// TwinCAT 3 PLC project Nepionic_PackML
// Title: Nepionic_PackML
// Company: Nepionic
// Author: Nepionic
// ProjectVersion: 0.1.0
// ProgramVersion: 3.1.4026.19
// libraries:
//   Tc2_System, * (Beckhoff Automation GmbH)
// project tree:
//   Commands/ AbortedCommands.TcIO, AbortingCommands.TcIO, ClearingCommands.TcIO, CompletedCommands.TcIO, CompletingCommands.TcIO, ExecuteCommands.TcIO, HeldCommands.TcIO, HoldingCommands.TcIO, IdleCommands.TcIO, ResettingCommands.TcIO, StartingCommands.TcIO, StoppedCommands.TcIO, StoppingCommands.TcIO, SuspendedCommands.TcIO, SuspendingCommands.TcIO, UnholdingCommands.TcIO, UnsuspendingCommands.TcIO
//   StateMachine/ State.TcDUT, StateMachine.TcPOU
//   UnitMode/ UnitMode.TcIO (not stored), DefaultUnitMode.TcPOU

// ---- StateMachine/State.TcDUT
{attribute 'qualified_only'}
{attribute 'strict'}
TYPE State :
(
	UNDEFINED := 0,
    CLEARING := 1,
    STOPPED := 2,
    STARTING := 3,
    IDLE := 4,
    SUSPENDED := 5,
	EXECUTE := 6,
    STOPPING := 7,
    ABORTING := 8,
    ABORTED := 9,
    HOLDING := 10,
    HELD := 11,
    UNHOLDING := 12,
    SUSPENDING := 13,
    UNSUSPENDING := 14,
    RESETTING := 15,
    COMPLETING := 16,
    COMPLETE := 17
);
END_TYPE

// ---- Commands/AbortedCommands.TcIO
INTERFACE PUBLIC AbortedCommands

METHOD PUBLIC Clear
END_METHOD

END_INTERFACE

// ---- Commands/AbortingCommands.TcIO
INTERFACE PUBLIC AbortingCommands

METHOD PUBLIC StateComplete
END_METHOD

END_INTERFACE

// ---- Commands/ClearingCommands.TcIO
INTERFACE PUBLIC ClearingCommands

METHOD PUBLIC Abort
END_METHOD

METHOD PUBLIC StateComplete
END_METHOD

END_INTERFACE

// ---- Commands/CompletedCommands.TcIO
INTERFACE PUBLIC CompletedCommands

METHOD PUBLIC Abort
END_METHOD

METHOD PUBLIC Reset
END_METHOD

METHOD PUBLIC Stop
END_METHOD

END_INTERFACE

// ---- Commands/CompletingCommands.TcIO
INTERFACE PUBLIC CompletingCommands

METHOD PUBLIC Abort
END_METHOD

METHOD PUBLIC StateComplete
END_METHOD

METHOD PUBLIC Stop
END_METHOD

END_INTERFACE

// ---- Commands/ExecuteCommands.TcIO
INTERFACE PUBLIC ExecuteCommands

METHOD PUBLIC Abort
END_METHOD

METHOD PUBLIC Hold
END_METHOD

METHOD PUBLIC StateComplete
END_METHOD

METHOD PUBLIC Stop
END_METHOD

METHOD PUBLIC Suspend
END_METHOD

END_INTERFACE

// ---- Commands/HeldCommands.TcIO
INTERFACE PUBLIC HeldCommands

METHOD PUBLIC Abort
END_METHOD

METHOD PUBLIC Stop
END_METHOD

METHOD PUBLIC Unhold
END_METHOD

END_INTERFACE

// ---- Commands/HoldingCommands.TcIO
INTERFACE PUBLIC HoldingCommands

METHOD PUBLIC Abort
END_METHOD

METHOD PUBLIC StateComplete
END_METHOD

METHOD PUBLIC Stop
END_METHOD

END_INTERFACE

// ---- Commands/IdleCommands.TcIO
INTERFACE PUBLIC IdleCommands

METHOD PUBLIC Abort
END_METHOD

METHOD PUBLIC Start
END_METHOD

METHOD PUBLIC Stop
END_METHOD

END_INTERFACE

// ---- Commands/ResettingCommands.TcIO
INTERFACE PUBLIC ResettingCommands

METHOD PUBLIC Abort
END_METHOD

METHOD PUBLIC StateComplete
END_METHOD

METHOD PUBLIC Stop
END_METHOD

END_INTERFACE

// ---- Commands/StartingCommands.TcIO
INTERFACE PUBLIC StartingCommands

METHOD PUBLIC Abort
END_METHOD

METHOD PUBLIC StateComplete
END_METHOD

END_INTERFACE

// ---- Commands/StoppedCommands.TcIO
INTERFACE StoppedCommands

METHOD PUBLIC Reset
END_METHOD

END_INTERFACE

// ---- Commands/StoppingCommands.TcIO
INTERFACE PUBLIC StoppingCommands

METHOD PUBLIC StateComplete
END_METHOD

END_INTERFACE

// ---- Commands/SuspendedCommands.TcIO
INTERFACE PUBLIC SuspendedCommands

METHOD PUBLIC Abort
END_METHOD

METHOD PUBLIC Stop
END_METHOD

METHOD PUBLIC Unsuspend
END_METHOD

END_INTERFACE

// ---- Commands/SuspendingCommands.TcIO
INTERFACE PUBLIC SuspendingCommands

METHOD PUBLIC Abort
END_METHOD

METHOD PUBLIC StateComplete
END_METHOD

METHOD PUBLIC Stop
END_METHOD

END_INTERFACE

// ---- Commands/UnholdingCommands.TcIO
INTERFACE PUBLIC UnholdingCommands

METHOD PUBLIC Abort
END_METHOD

METHOD PUBLIC StateComplete
END_METHOD

METHOD PUBLIC Stop
END_METHOD

END_INTERFACE

// ---- Commands/UnsuspendingCommands.TcIO
INTERFACE PUBLIC UnsuspendingCommands

METHOD PUBLIC Abort
END_METHOD

METHOD PUBLIC StateComplete
END_METHOD

METHOD PUBLIC Stop
END_METHOD

END_INTERFACE

// ---- StateMachine/StateMachine.TcPOU
{attribute 'linkalways'} 
{attribute 'no_explicit_call' := 'This FB is a CLASS and must be accessed using methods or properties'}
{attribute 'enable_dynamic_creation'}
FUNCTION_BLOCK PUBLIC StateMachine
VAR_GENERIC CONSTANT
	initial_state : State := State.Idle;
END_VAR
IMPLEMENTS
	AbortingCommands,
	ClearingCommands,
	HeldCommands,
	CompletingCommands,
	ExecuteCommands,
	AbortedCommands,
	CompletedCommands,
	HoldingCommands,
	UnsuspendingCommands,
	UnholdingCommands,
	SuspendingCommands,
	SuspendedCommands,
	IdleCommands,
	ResettingCommands,
	StartingCommands,
	StoppedCommands,
	StoppingCommands
VAR
	current_state : State := initial_state;
END_VAR

METHOD PUBLIC Abort
IF IsAborting OR IsAborted THEN
	RETURN;
END_IF

LogCommand('Abort');
ChangeState(State.Aborting);
END_METHOD

METHOD PRIVATE ChangeState
VAR_INPUT
	state : State;
END_VAR
ExitingState(current_state);
current_state := state;
EnteringState(current_state);
END_METHOD

METHOD PUBLIC Clear
IF IsAborted THEN
	LogCommand('Clear');
	ChangeState(State.Clearing);
END_IF
END_METHOD

{attribute 'monitoring':='call'}
PROPERTY PUBLIC CurrentState : State
GET
CurrentState := current_state;
END_GET
END_PROPERTY

METHOD PRIVATE EnteringState
VAR_INPUT
	state : State;
END_VAR
VAR
	state_string : STRING;
END_VAR
state_string := TO_STRING(state);
END_METHOD

METHOD PRIVATE ExitingState
VAR_INPUT
	state : State;
END_VAR
VAR
	state_string : STRING;
END_VAR
state_string := TO_STRING(state);
END_METHOD

METHOD PUBLIC Hold
IF IsExecuting THEN
	LogCommand('Hold');
	ChangeState(State.Holding);
END_IF
END_METHOD

{attribute 'monitoring':='call'}
PROPERTY PUBLIC IsAborted : BOOL
GET
IsAborted := (current_state = State.Aborted);
END_GET
END_PROPERTY

{attribute 'monitoring':='call'}
PROPERTY PUBLIC IsAborting : BOOL
GET
IsAborting := (current_state = State.Aborting);
END_GET
END_PROPERTY

{attribute 'monitoring':='call'}
PROPERTY PUBLIC IsClearing : BOOL
GET
IsClearing := (current_state = State.Clearing);
END_GET
END_PROPERTY

{attribute 'monitoring':='call'}
PROPERTY PUBLIC IsCompleted : BOOL
GET
IsCompleted := (current_state = State.Completed);
END_GET
END_PROPERTY

{attribute 'monitoring':='call'}
PROPERTY PUBLIC IsCompleting : BOOL
GET
IsCompleting := (current_state = State.Completing);
END_GET
END_PROPERTY

{attribute 'monitoring':='call'}
PROPERTY PUBLIC IsExecuting : BOOL
GET
IsExecuting := (current_state = State.Execute);
END_GET
END_PROPERTY

{attribute 'monitoring':='call'}
PROPERTY PUBLIC IsHeld : BOOL
GET
IsHeld := (current_state = State.Held);
END_GET
END_PROPERTY

{attribute 'monitoring':='call'}
PROPERTY PUBLIC IsHolding : BOOL
GET
IsHolding := (current_state = State.Holding);
END_GET
END_PROPERTY

{attribute 'monitoring':='call'}
PROPERTY PUBLIC IsIdle : BOOL
GET
isIdle := (current_state = State.Idle);
END_GET
END_PROPERTY

{attribute 'monitoring':='call'}
PROPERTY PUBLIC IsResetting : BOOL
GET
IsResetting := (current_state = State.Resetting);
END_GET
END_PROPERTY

{attribute 'monitoring':='call'}
PROPERTY PUBLIC IsStarting : BOOL
GET
IsStarting := (current_state = State.Starting);
END_GET
END_PROPERTY

{attribute 'monitoring':='call'}
PROPERTY PUBLIC IsStopped : BOOL
GET
isStopped := (current_state = State.Stopped);
END_GET
END_PROPERTY

{attribute 'monitoring':='call'}
PROPERTY PUBLIC IsStopping : BOOL
GET
IsStopping := (current_state = State.Stopping);
END_GET
END_PROPERTY

{attribute 'monitoring':='call'}
PROPERTY PUBLIC IsSuspended : BOOL
GET
IsSuspended := (current_state = State.Suspended);
END_GET
END_PROPERTY

{attribute 'monitoring':='call'}
PROPERTY PUBLIC IsSuspending : BOOL
GET
IsSuspending := (current_state = State.Suspending);
END_GET
END_PROPERTY

{attribute 'monitoring':='call'}
PROPERTY PUBLIC IsUnholding : BOOL
GET
IsUnholding := (current_state = State.Unholding);
END_GET
END_PROPERTY

{attribute 'monitoring':='call'}
PROPERTY PUBLIC IsUnsuspending : BOOL
GET
IsUnsuspending := (current_state = State.Unsuspending);
END_GET
END_PROPERTY

METHOD PRIVATE LogCommand
VAR_INPUT
	command : STRING;
END_VAR
END_METHOD

METHOD PUBLIC Reset
IF IsStopped OR IsCompleted THEN
	LogCommand('Reset');
	ChangeState(State.Resetting);
END_IF
END_METHOD

METHOD PUBLIC Start
IF IsIdle THEN
	LogCommand('Start');
	ChangeState(State.Starting);
END_IF
END_METHOD

METHOD PUBLIC StateComplete
CASE current_state OF 
	State.Idle:
		RETURN;
	
	State.Starting:
		ChangeState(State.Execute);
		
	State.Execute:
		ChangeState(State.Completing);
		
	State.Completing:
		ChangeState(State.Completed);
	
	State.Completed:
		RETURN;
	
	State.Stopping:
		ChangeState(State.Stopped);
	
	State.Stopped:
		RETURN;
	
	State.Resetting:
		ChangeState(State.Idle);
	
	State.Holding:
		ChangeState(State.Held);
	
	State.Held:
		RETURN;
	
	State.Unholding:
		ChangeState(State.Execute);
	
	State.Suspending:
		ChangeState(State.Suspended);
	
	State.Suspended:
		RETURN;
	
	State.Unsuspending:
		ChangeState(State.Execute);
	
	State.Clearing:
		ChangeState(State.Stopped);
	
	State.Aborted:
		RETURN;
	
	State.Aborting:
		ChangeState(State.Aborted);
END_CASE

LogCommand('StateComplete');
END_METHOD

METHOD PUBLIC Stop
CASE current_state OF
	State.Stopped: RETURN;
	State.Stopping: RETURN;
	State.Clearing: RETURN;
	State.Aborted: RETURN;
	State.Aborting: RETURN;
END_CASE

LogCommand('Stop');
ChangeState(State.Stopping);
END_METHOD

METHOD PUBLIC Suspend
IF IsExecuting THEN 
	LogCommand('Suspend');
	ChangeState(State.Suspending);
END_IF
END_METHOD

METHOD PUBLIC Unhold
IF IsHeld THEN
	LogCommand('Unhold');
	ChangeState(State.Unholding);
END_IF
END_METHOD

METHOD PUBLIC Unsuspend
IF IsSuspended THEN
	LogCommand('Unsuspend');
	ChangeState(State.Unsuspending);
END_IF
END_METHOD

END_FUNCTION_BLOCK

// ---- UnitMode/DefaultUnitMode.TcPOU
{attribute 'linkalways'} 
{attribute 'no_explicit_call' := 'This FB is a CLASS and must be accessed using methods or properties'}
{attribute 'enable_dynamic_creation'}
FUNCTION_BLOCK PUBLIC ABSTRACT DefaultUnitMode
VAR_GENERIC CONSTANT
	initial_state : State := State.Idle;
END_VAR
IMPLEMENTS UnitMode
VAR
	state_machine : StateMachine<initial_state>;
END_VAR

METHOD PUBLIC Abort
state_machine.Abort();
END_METHOD

METHOD PROTECTED Aborted
VAR_INPUT
	commands : AbortedCommands;
END_VAR
END_METHOD

METHOD PROTECTED Aborting
VAR_INPUT
	commands : AbortingCommands;
END_VAR
commands.StateComplete();
END_METHOD

METHOD PUBLIC Clear
state_machine.Clear();
END_METHOD

METHOD PROTECTED Clearing
VAR_INPUT
	commands : ClearingCommands;
END_VAR
commands.StateComplete();
END_METHOD

METHOD PROTECTED Completed
VAR_INPUT
	commands : CompletedCommands;
END_VAR
END_METHOD

METHOD PROTECTED Completing
VAR_INPUT
	commands : CompletingCommands;
END_VAR
commands.StateComplete();
END_METHOD

{attribute 'monitoring':='call'}
PROPERTY PUBLIC CurrentState : State
GET
CurrentState := state_machine.CurrentState;
END_GET
END_PROPERTY

METHOD PUBLIC CyclicCall
IF state_machine.IsIdle THEN 
	Idle(state_machine);
END_IF

IF state_machine.IsStarting THEN
	Starting(state_machine);
END_IF

IF state_machine.IsExecuting THEN
	Execute(state_machine);
END_IF

IF state_machine.IsCompleting THEN
	Completing(state_machine);
END_IF

IF state_machine.IsCompleted THEN
	Completed(state_machine);
END_IF

IF state_machine.IsStopping THEN
	Stopping(state_machine);
END_IF

IF state_machine.IsStopped THEN
	Stopped(state_machine);
END_IF

IF state_machine.IsResetting THEN
	Resetting(state_machine);
END_IF

IF state_machine.IsHolding THEN
	Holding(state_machine);
END_IF

IF state_machine.IsHeld THEN
	Held(state_machine);
END_IF

IF state_machine.IsUnholding THEN
	Unholding(state_machine);
END_IF

IF state_machine.IsSuspending THEN
	Suspending(state_machine);
END_IF

IF state_machine.IsSuspended THEN
	Suspended(state_machine);
END_IF

IF state_machine.IsUnsuspending THEN
	Unsuspending(state_machine);
END_IF

IF state_machine.IsClearing THEN
	Clearing(state_machine);
END_IF

IF state_machine.IsAborted THEN
	Aborted(state_machine);
END_IF

IF state_machine.IsAborting THEN
	Aborting(state_machine);
END_IF
END_METHOD

METHOD PROTECTED Execute
VAR_INPUT
	commands : ExecuteCommands;
END_VAR
commands.StateComplete();
END_METHOD

METHOD PROTECTED Held
VAR_INPUT
	commands : HeldCommands;
END_VAR
END_METHOD

METHOD PUBLIC Hold
state_machine.Hold();
END_METHOD

METHOD PROTECTED Holding
VAR_INPUT
	commands : HoldingCommands;
END_VAR
commands.StateComplete();
END_METHOD

METHOD PROTECTED Idle
VAR_INPUT
	commands : IdleCommands;
END_VAR
END_METHOD

{attribute 'monitoring':='call'}
PROPERTY PUBLIC IsAborted : bool
GET
IsAborted := state_machine.IsAborted;
END_GET
END_PROPERTY

{attribute 'monitoring':='call'}
PROPERTY PUBLIC IsAborting : bool
GET
IsAborting := state_machine.IsAborting;
END_GET
END_PROPERTY

{attribute 'monitoring':='call'}
PROPERTY PUBLIC IsClearing : bool
GET
IsClearing := state_machine.IsClearing;
END_GET
END_PROPERTY

{attribute 'monitoring':='call'}
PROPERTY PUBLIC IsCompleted : bool
GET
IsCompleted := state_machine.IsCompleted;
END_GET
END_PROPERTY

{attribute 'monitoring':='call'}
PROPERTY PUBLIC IsCompleting : bool
GET
IsCompleting := state_machine.IsCompleting;
END_GET
END_PROPERTY

{attribute 'monitoring':='call'}
PROPERTY PUBLIC IsExecuting : bool
GET
IsExecuting := state_machine.IsExecuting;
END_GET
END_PROPERTY

{attribute 'monitoring':='call'}
PROPERTY PUBLIC IsHeld : bool
GET
IsHeld := state_machine.IsHeld;
END_GET
END_PROPERTY

{attribute 'monitoring':='call'}
PROPERTY PUBLIC IsHolding : bool
GET
IsHolding := state_machine.IsHolding;
END_GET
END_PROPERTY

{attribute 'monitoring':='call'}
PROPERTY PUBLIC IsIdle : BOOL
GET
isIdle := state_machine.isIdle;
END_GET
END_PROPERTY

{attribute 'monitoring':='call'}
PROPERTY PUBLIC IsResetting : bool
GET
IsResetting := state_machine.IsResetting;
END_GET
END_PROPERTY

{attribute 'monitoring':='call'}
PROPERTY PUBLIC IsStarting : bool
GET
IsStarting := state_machine.IsStarting;
END_GET
END_PROPERTY

{attribute 'monitoring':='call'}
PROPERTY PUBLIC IsStopped : BOOL
GET
isStopped := state_machine.isStopped;
END_GET
END_PROPERTY

{attribute 'monitoring':='call'}
PROPERTY PUBLIC IsStopping : bool
GET
IsStopping := state_machine.IsStopping;
END_GET
END_PROPERTY

{attribute 'monitoring':='call'}
PROPERTY PUBLIC IsSuspended : bool
GET
IsSuspended := state_machine.IsSuspended;
END_GET
END_PROPERTY

{attribute 'monitoring':='call'}
PROPERTY PUBLIC IsSuspending : bool
GET
IsSuspending := state_machine.IsSuspending;
END_GET
END_PROPERTY

{attribute 'monitoring':='call'}
PROPERTY PUBLIC IsUnholding : bool
GET
IsUnholding := state_machine.IsUnholding;
END_GET
END_PROPERTY

{attribute 'monitoring':='call'}
PROPERTY PUBLIC IsUnsuspending : bool
GET
IsUnsuspending := state_machine.IsUnsuspending;
END_GET
END_PROPERTY

METHOD PUBLIC Reset
state_machine.Reset();
END_METHOD

METHOD PROTECTED Resetting
VAR_INPUT
	commands : ResettingCommands;
END_VAR
commands.StateComplete();
END_METHOD

METHOD PUBLIC Start
state_machine.Start();
END_METHOD

METHOD PROTECTED Starting
VAR_INPUT
	commands : StartingCommands;
END_VAR
commands.StateComplete();
END_METHOD

METHOD PUBLIC Stop
state_machine.Stop();
END_METHOD

METHOD PROTECTED Stopped
VAR_INPUT
	commands : StoppedCommands;
END_VAR
END_METHOD

METHOD PROTECTED Stopping
VAR_INPUT
	commands : StoppingCommands;
END_VAR
commands.StateComplete();
END_METHOD

METHOD PUBLIC Suspend
state_machine.Suspend();
END_METHOD

METHOD PROTECTED Suspended
VAR_INPUT
	commands : SuspendedCommands;
END_VAR
END_METHOD

METHOD PROTECTED Suspending
VAR_INPUT
	commands : SuspendingCommands;
END_VAR
commands.StateComplete();
END_METHOD

METHOD PUBLIC Unhold
state_machine.Unhold();
END_METHOD

METHOD PROTECTED Unholding
VAR_INPUT
	commands : UnholdingCommands;
END_VAR
commands.StateComplete();
END_METHOD

METHOD PUBLIC Unsuspend
state_machine.Unsuspend();
END_METHOD

METHOD PROTECTED Unsuspending
VAR_INPUT
	commands : UnsuspendingCommands;
END_VAR
commands.StateComplete();
END_METHOD

END_FUNCTION_BLOCK
